FUNCTION_BLOCK Test_F_UDINT_TO_DINT_Conversion EXTENDS T_UnitTestBase
VAR
    InputValue     : UDINT;
    ConvertedValue : DINT;
END_VAR

{attribute 'analysis' := '-33'} // inhibit unused variable warning
METHOD RunTest
IF Retest THEN
    SUPER^.Init();
END_IF

IF TestCompleted THEN
    RETURN;
END_IF

F_Inc(CycleCount);
IF CycleCount > 1000 THEN
    Fail(Message := 'Timeout');
END_IF

InputValue     := UDINT#2147483648;            // too big
ConvertedValue := F_UDINT_TO_DINT(InputValue); // limit to largest DINT

AssertIsTrue(Condition := (ConvertedValue = 2147483647),
             Message   := 'F_UDINT_TO_DINT returns incorrect value');

TestCompleted := TRUE;
END_METHOD

END_FUNCTION_BLOCK

(* stored: Version 1.1.0.1, ProductVersion 3.1.4024.15
   POU Test_F_UDINT_TO_DINT_Conversion: Id {0f7dcc90-c1e5-4697-8983-52848bcba636}, SpecialFunc None
   Method RunTest: Id {4aeb1853-9057-45ad-afb4-122c04cd546c} *)
